{attribute 'OPC.UA.DA' := '1'}
TYPE IoSJH108A :
STRUCT					
	OutputOpenAirValve	AT %Q* : BOOL;	
	OutputStaticEliminationInterrupt AT %Q* : BOOL;
END_STRUCT
END_TYPE

(* stored: Version 1.1.0.1, ProductVersion 3.1.4024.12
   DUT IoSJH108A: Id {64df1686-9c72-4375-9ade-c239d5c012dc} *)
